% RSLogix 500 project PUMP PROTECTION.RSS, saved by version 8.30.00.16 %
PROJECT "UNTITLED"    % processor: Bul.1763 MicroLogix 1100 Series B %

PROGRAM FILES
  LAD 2 "MAIN"  6 rungs
  LAD 3 "OUTPUT"  4 rungs
  LAD 4 "INPUT"  5 rungs
  LAD 5 "CONTROLS"  6 rungs
  LAD 6 "ALARMS"  8 rungs
  LAD 7 "HOA"  6 rungs

DATA FILES
  O0 OUTPUT  4 elements
  I1 INPUT  6 elements
  S2 STATUS  66 elements
  B3 BINARY  3 elements
  T4 TIMER  4 elements
  C5 COUNTER  1 elements
  R6 CONTROL  1 elements
  N7 INTEGER  10 elements
  F8 FLOAT  1 elements

LADDER 2 "MAIN"
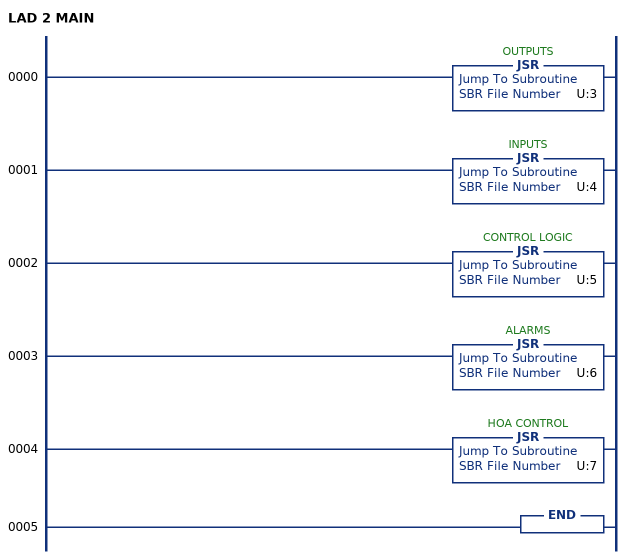
% Rung: 0 %
SOR JSR U:3 EOR
%   U:3  "OUTPUTS" %
% Rung: 1 %
SOR JSR U:4 EOR
%   U:4  "INPUTS" %
% Rung: 2 %
SOR JSR U:5 EOR
%   U:5  "CONTROL LOGIC" %
% Rung: 3 %
SOR JSR U:6 EOR
%   U:6  "ALARMS" %
% Rung: 4 %
SOR JSR U:7 EOR
%   U:7  "HOA CONTROL" %
% Rung: 5 %
SOR END EOR

LADDER 3 "OUTPUT"
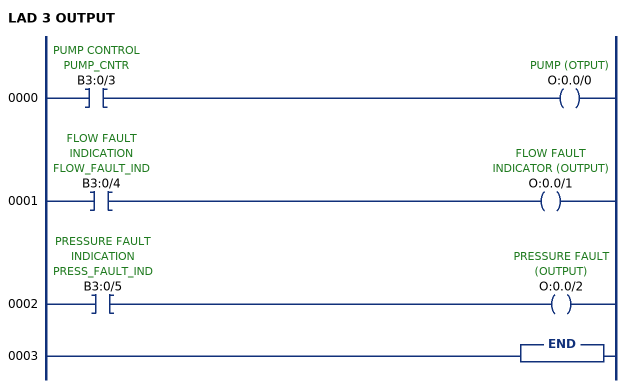
% Rung: 0 %
SOR XIC B3:0/3 OTE O:0.0/0 EOR
%   B3:0/3  PUMP_CNTR  "PUMP CONTROL" %
%   O:0.0/0  "PUMP (OTPUT)" %
% Rung: 1 %
SOR XIC B3:0/4 OTE O:0.0/1 EOR
%   B3:0/4  FLOW_FAULT_IND  "FLOW FAULT INDICATION" %
%   O:0.0/1  "FLOW FAULT INDICATOR (OUTPUT)" %
% Rung: 2 %
SOR XIC B3:0/5 OTE O:0.0/2 EOR
%   B3:0/5  PRESS_FAULT_IND  "PRESSURE FAULT INDICATION" %
%   O:0.0/2  "PRESSURE FAULT (OUTPUT)" %
% Rung: 3 %
SOR END EOR

LADDER 4 "INPUT"
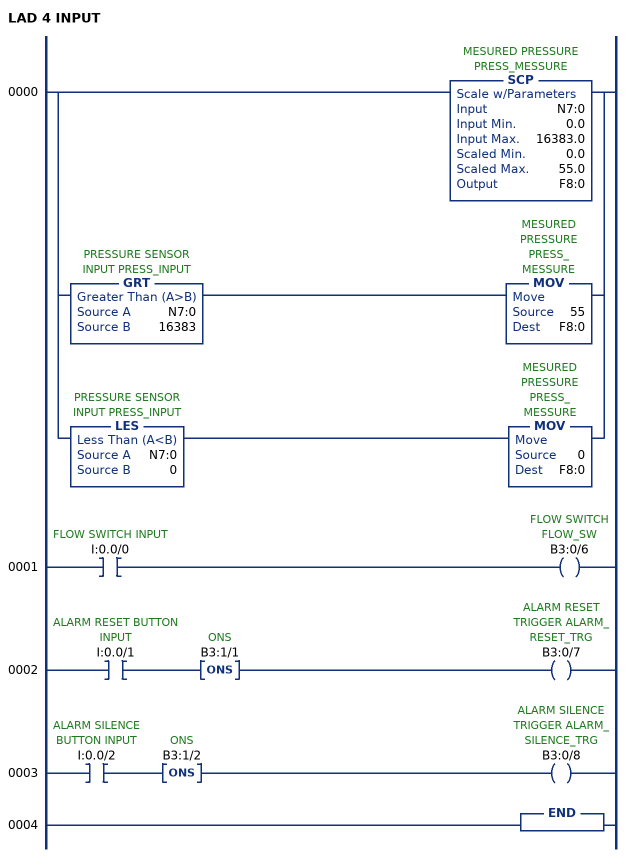
% Rung: 0 %
SOR BST SCP N7:0 0.0 16383.0 0.0 55.0 F8:0 NXB GRT N7:0 16383 MOV 55 F8:0 NXB LES N7:0 0 MOV 0 F8:0 BND EOR
%   N7:0  PRESS_INPUT  "PRESSURE SENSOR INPUT" %
%   F8:0  PRESS_MESSURE  "MESURED PRESSURE" %
% Rung: 1 %
SOR XIC I:0.0/0 OTE B3:0/6 EOR
%   I:0.0/0  "FLOW SWITCH INPUT" %
%   B3:0/6  FLOW_SW  "FLOW SWITCH" %
% Rung: 2 %
SOR XIC I:0.0/1 ONS B3:1/1 OTE B3:0/7 EOR
%   I:0.0/1  "ALARM RESET BUTTON INPUT" %
%   B3:1/1  "ONS" %
%   B3:0/7  ALARM_RESET_TRG  "ALARM RESET TRIGGER" %
% Rung: 3 %
SOR XIC I:0.0/2 ONS B3:1/2 OTE B3:0/8 EOR
%   I:0.0/2  "ALARM SILENCE BUTTON INPUT" %
%   B3:1/2  "ONS" %
%   B3:0/8  ALARM_SILENCE_TRG  "ALARM SILENCE TRIGGER" %
% Rung: 4 %
SOR END EOR

LADDER 5 "CONTROLS"
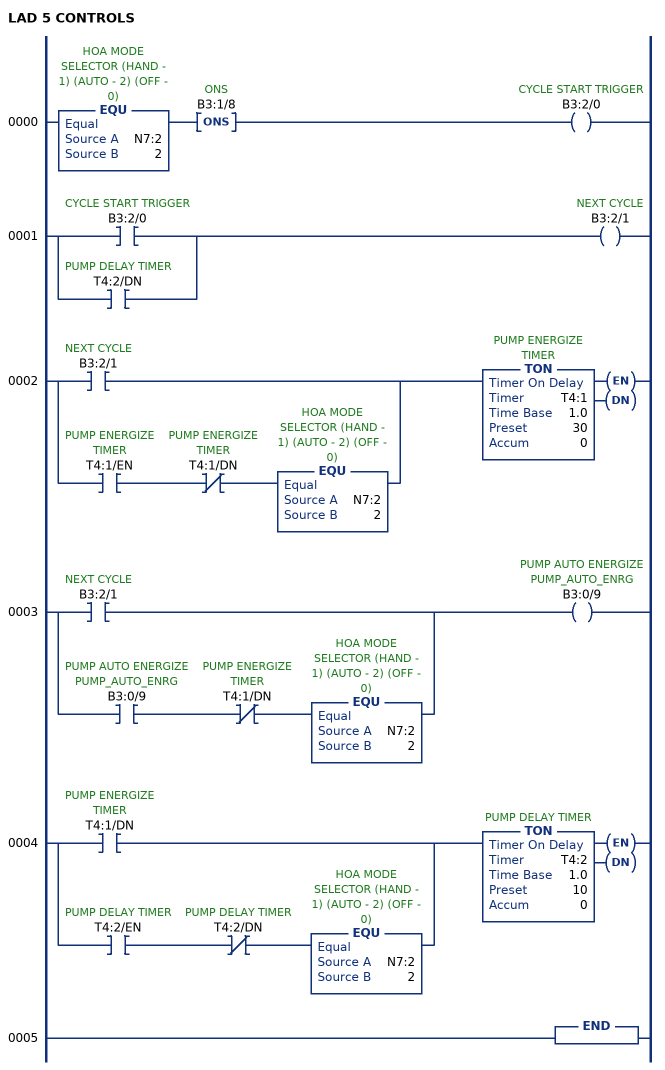
% Rung: 0 %
SOR EQU N7:2 2 ONS B3:1/8 OTE B3:2/0 EOR
%   N7:2  "HOA MODE SELECTOR (HAND - 1) (AUTO - 2) (OFF - 0)" %
%   B3:1/8  "ONS" %
%   B3:2/0  "CYCLE START TRIGGER" %
% Rung: 1 %
SOR BST XIC B3:2/0 NXB XIC T4:2/DN BND OTE B3:2/1 EOR
%   B3:2/0  "CYCLE START TRIGGER" %
%   T4:2  "PUMP DELAY TIMER" %
%   B3:2/1  "NEXT CYCLE" %
% Rung: 2 %
SOR BST XIC B3:2/1 NXB XIC T4:1/EN XIO T4:1/DN EQU N7:2 2 BND TON T4:1 1.0 30 0 EOR
%   B3:2/1  "NEXT CYCLE" %
%   T4:1  "PUMP ENERGIZE TIMER" %
%   N7:2  "HOA MODE SELECTOR (HAND - 1) (AUTO - 2) (OFF - 0)" %
% Rung: 3 %
SOR BST XIC B3:2/1 NXB XIC B3:0/9 XIO T4:1/DN EQU N7:2 2 BND OTE B3:0/9 EOR
%   B3:2/1  "NEXT CYCLE" %
%   B3:0/9  PUMP_AUTO_ENRG  "PUMP AUTO ENERGIZE" %
%   T4:1  "PUMP ENERGIZE TIMER" %
%   N7:2  "HOA MODE SELECTOR (HAND - 1) (AUTO - 2) (OFF - 0)" %
% Rung: 4 %
SOR BST XIC T4:1/DN NXB XIC T4:2/EN XIO T4:2/DN EQU N7:2 2 BND TON T4:2 1.0 10 0 EOR
%   T4:1  "PUMP ENERGIZE TIMER" %
%   T4:2  "PUMP DELAY TIMER" %
%   N7:2  "HOA MODE SELECTOR (HAND - 1) (AUTO - 2) (OFF - 0)" %
% Rung: 5 %
SOR END EOR

LADDER 6 "ALARMS"
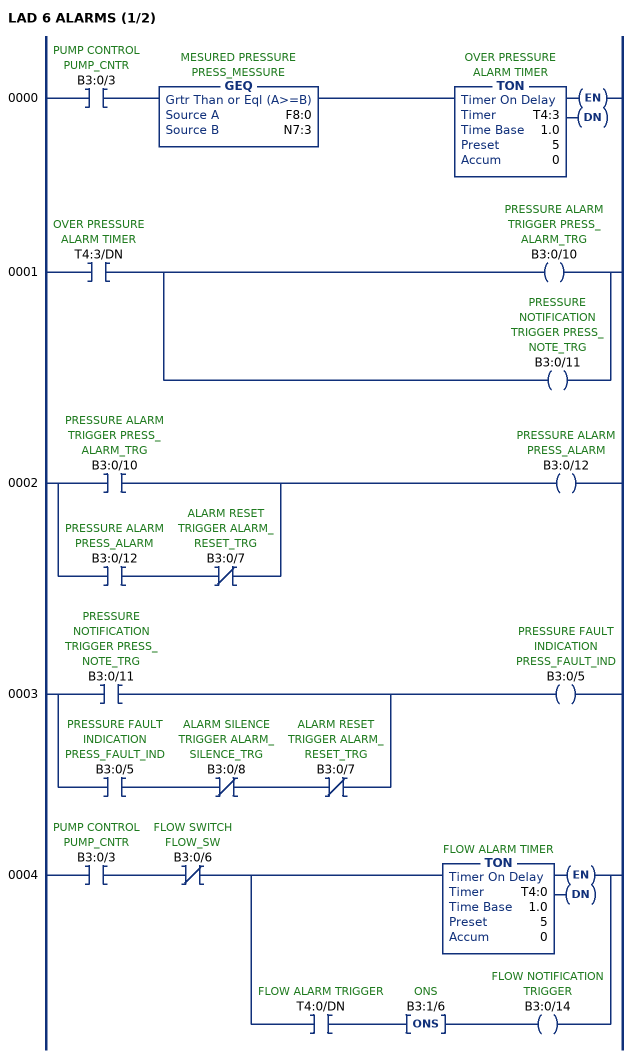
% Rung: 0 %
SOR XIC B3:0/3 GEQ F8:0 N7:3 TON T4:3 1.0 5 0 EOR
%   B3:0/3  PUMP_CNTR  "PUMP CONTROL" %
%   F8:0  PRESS_MESSURE  "MESURED PRESSURE" %
%   N7:3  "PRESSURE LEVEL THRESHOLD" %
%   T4:3  "OVER PRESSURE ALARM TIMER" %
% Rung: 1 %
SOR XIC T4:3/DN BST OTE B3:0/10 NXB OTE B3:0/11 BND EOR
%   T4:3  "OVER PRESSURE ALARM TIMER" %
%   B3:0/10  PRESS_ALARM_TRG  "PRESSURE ALARM TRIGGER" %
%   B3:0/11  PRESS_NOTE_TRG  "PRESSURE NOTIFICATION TRIGGER" %
% Rung: 2 %
SOR BST XIC B3:0/10 NXB XIC B3:0/12 XIO B3:0/7 BND OTE B3:0/12 EOR
%   B3:0/10  PRESS_ALARM_TRG  "PRESSURE ALARM TRIGGER" %
%   B3:0/12  PRESS_ALARM  "PRESSURE ALARM" %
%   B3:0/7  ALARM_RESET_TRG  "ALARM RESET TRIGGER" %
% Rung: 3 %
SOR BST XIC B3:0/11 NXB XIC B3:0/5 XIO B3:0/8 XIO B3:0/7 BND OTE B3:0/5 EOR
%   B3:0/11  PRESS_NOTE_TRG  "PRESSURE NOTIFICATION TRIGGER" %
%   B3:0/5  PRESS_FAULT_IND  "PRESSURE FAULT INDICATION" %
%   B3:0/8  ALARM_SILENCE_TRG  "ALARM SILENCE TRIGGER" %
%   B3:0/7  ALARM_RESET_TRG  "ALARM RESET TRIGGER" %
% Rung: 4 %
SOR XIC B3:0/3 XIO B3:0/6 BST TON T4:0 1.0 5 0 NXB XIC T4:0/DN ONS B3:1/6 OTE B3:0/14 BND EOR
%   B3:0/3  PUMP_CNTR  "PUMP CONTROL" %
%   B3:0/6  FLOW_SW  "FLOW SWITCH" %
%   T4:0  "FLOW ALARM TIMER" %
%   T4:0/DN  "FLOW ALARM TRIGGER" %
%   B3:1/6  "ONS" %
%   B3:0/14  "FLOW NOTIFICATION TRIGGER" %

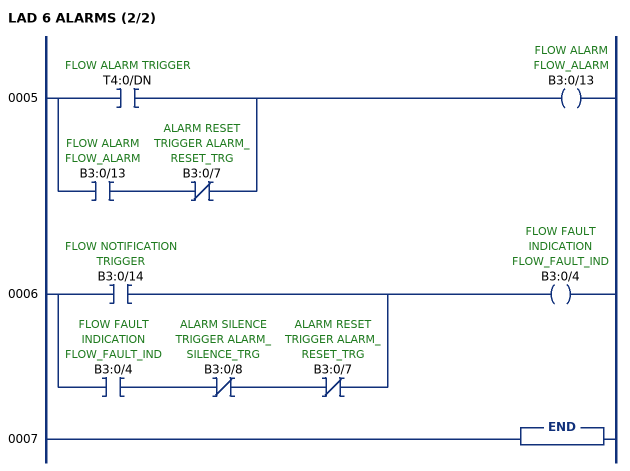
% Rung: 5 %
SOR BST XIC T4:0/DN NXB XIC B3:0/13 XIO B3:0/7 BND OTE B3:0/13 EOR
%   T4:0/DN  "FLOW ALARM TRIGGER" %
%   B3:0/13  FLOW_ALARM  "FLOW ALARM" %
%   B3:0/7  ALARM_RESET_TRG  "ALARM RESET TRIGGER" %
% Rung: 6 %
SOR BST XIC B3:0/14 NXB XIC B3:0/4 XIO B3:0/8 XIO B3:0/7 BND OTE B3:0/4 EOR
%   B3:0/14  "FLOW NOTIFICATION TRIGGER" %
%   B3:0/4  FLOW_FAULT_IND  "FLOW FAULT INDICATION" %
%   B3:0/8  ALARM_SILENCE_TRG  "ALARM SILENCE TRIGGER" %
%   B3:0/7  ALARM_RESET_TRG  "ALARM RESET TRIGGER" %
% Rung: 7 %
SOR END EOR

LADDER 7 "HOA"
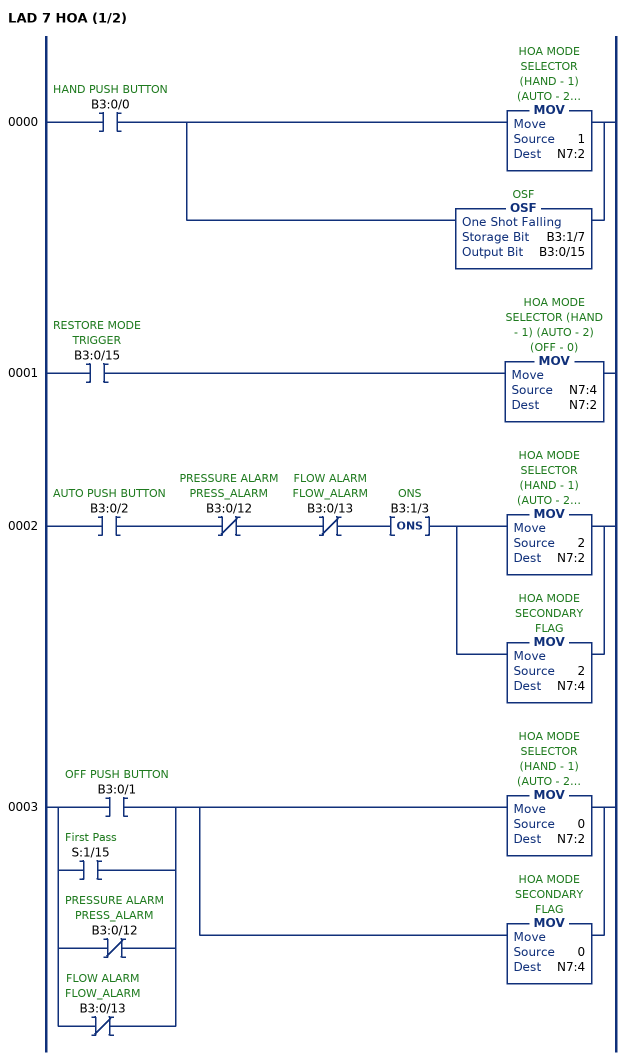
% Rung: 0 %
SOR XIC B3:0/0 BST MOV 1 N7:2 NXB OSF B3:1/7 B3:0/15 BND EOR
%   B3:0/0  "HAND PUSH BUTTON" %
%   N7:2  "HOA MODE SELECTOR (HAND - 1) (AUTO - 2) (OFF - 0)" %
%   B3:1/7  "OSF" %
%   B3:0/15  "RESTORE MODE TRIGGER" %
% Rung: 1 %
SOR XIC B3:0/15 MOV N7:4 N7:2 EOR
%   B3:0/15  "RESTORE MODE TRIGGER" %
%   N7:4  "HOA MODE SECONDARY FLAG" %
%   N7:2  "HOA MODE SELECTOR (HAND - 1) (AUTO - 2) (OFF - 0)" %
% Rung: 2 %
SOR XIC B3:0/2 XIO B3:0/12 XIO B3:0/13 ONS B3:1/3 BST MOV 2 N7:2 NXB MOV 2 N7:4 BND EOR
%   B3:0/2  "AUTO PUSH BUTTON" %
%   B3:0/12  PRESS_ALARM  "PRESSURE ALARM" %
%   B3:0/13  FLOW_ALARM  "FLOW ALARM" %
%   B3:1/3  "ONS" %
%   N7:2  "HOA MODE SELECTOR (HAND - 1) (AUTO - 2) (OFF - 0)" %
%   N7:4  "HOA MODE SECONDARY FLAG" %
% Rung: 3 %
SOR BST XIC B3:0/1 NXB XIC S:1/15 NXB XIO B3:0/12 NXB XIO B3:0/13 BND BST MOV 0 N7:2 NXB MOV 0 N7:4 BND EOR
%   B3:0/1  "OFF PUSH BUTTON" %
%   S:1/15  "First Pass" %
%   B3:0/12  PRESS_ALARM  "PRESSURE ALARM" %
%   B3:0/13  FLOW_ALARM  "FLOW ALARM" %
%   N7:2  "HOA MODE SELECTOR (HAND - 1) (AUTO - 2) (OFF - 0)" %
%   N7:4  "HOA MODE SECONDARY FLAG" %

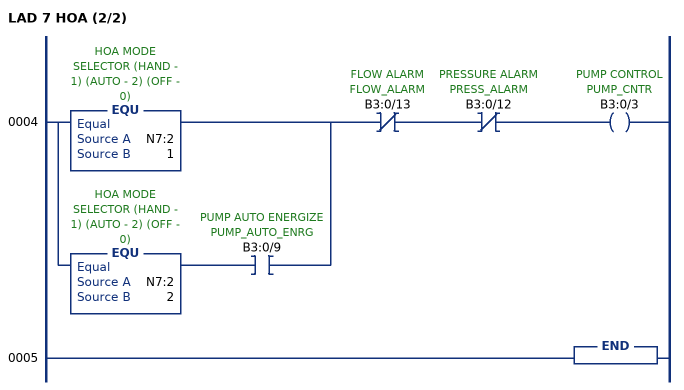
% Rung: 4 %
SOR BST EQU N7:2 1 NXB EQU N7:2 2 XIC B3:0/9 BND XIO B3:0/13 XIO B3:0/12 OTE B3:0/3 EOR
%   N7:2  "HOA MODE SELECTOR (HAND - 1) (AUTO - 2) (OFF - 0)" %
%   B3:0/9  PUMP_AUTO_ENRG  "PUMP AUTO ENERGIZE" %
%   B3:0/13  FLOW_ALARM  "FLOW ALARM" %
%   B3:0/12  PRESS_ALARM  "PRESSURE ALARM" %
%   B3:0/3  PUMP_CNTR  "PUMP CONTROL" %
% Rung: 5 %
SOR END EOR

OTHER DOCUMENTED ADDRESSES
  B3:0  "HAND PUSHBUTTON"
  B3:1/0  "ONS"
  B3:1/4  "ONS"
  B3:1/5  "ONS"
  B3:3  "AUTO PUSHBUTTON"
  N7:1  "PRESSURE SENSOR MESSURE"

DATA TABLE (non-zero values as saved)
DATA T4
% .PRE .ACC %
% T4:0 % 5 0
% T4:1 % 30 0
% T4:2 % 10 0
% T4:3 % 5 0
DATA N7
% N7:0 % 0 0 0 30 0 0 0 0 0 0
